INTERFACE I_ServoMotor

METHOD BeweegNaarDoel
VAR_INPUT
END_VAR
END_METHOD

PROPERTY DoelPositie : int
GET
END_GET
SET
END_SET
END_PROPERTY

PROPERTY Positie : int
GET
END_GET
END_PROPERTY

METHOD Start
VAR_INPUT
END_VAR
END_METHOD

METHOD Stop
VAR_INPUT
END_VAR
END_METHOD

END_INTERFACE

(* stored: Version 1.1.0.1
   Itf I_ServoMotor: Id {c243c482-42c3-4a76-81f1-ac3a4417e219}
   Method BeweegNaarDoel: Id {4f8b0714-7117-4f8d-913a-bddf18ac46d8}
   Property DoelPositie: Id {2f19f556-3609-47a6-b7da-5b4b1d4853bd}
   Get Get: Id {009ace2c-5c01-4643-b382-4715959ee1ac}
   Set Set: Id {3c8bf024-b765-4728-8adc-3950c46589a5}
   Property Positie: Id {d3d21827-b776-4526-9cf4-5b9802ab2987}
   Get Get: Id {9c055e2c-96fa-4e41-9eaf-6112a7c3e721}
   Method Start: Id {7f1b6655-17b0-4be9-9c56-a04be7b9ab23}
   Method Stop: Id {162c2817-abfe-4cc6-b2cb-cc3663fe1458} *)
